FUNCTION_BLOCK MGE (* Composite Function Block Type *)
  (* Standard: 61499-2 *)
  (* Version 0.9, 12/05/2026, Medidor Geral de Energia. CAT top-level com 2 SYMLINKMULTIVARDST do tipo base Runtime.System.SYMLINKMULTIVARDST (sem hash - EAE expande pelo InterfaceParams). SYMLINKMULTIVARDST1 = 16xREAL (tensoes/correntes/pot ativa parcial+total/pot reativa parcial); SYMLINKMULTIVARDST2 = 4xREAL (pot reativa total/freq/FP/pot aparente total). *)
  PACKAGE Hidryco.HidrycoLib;
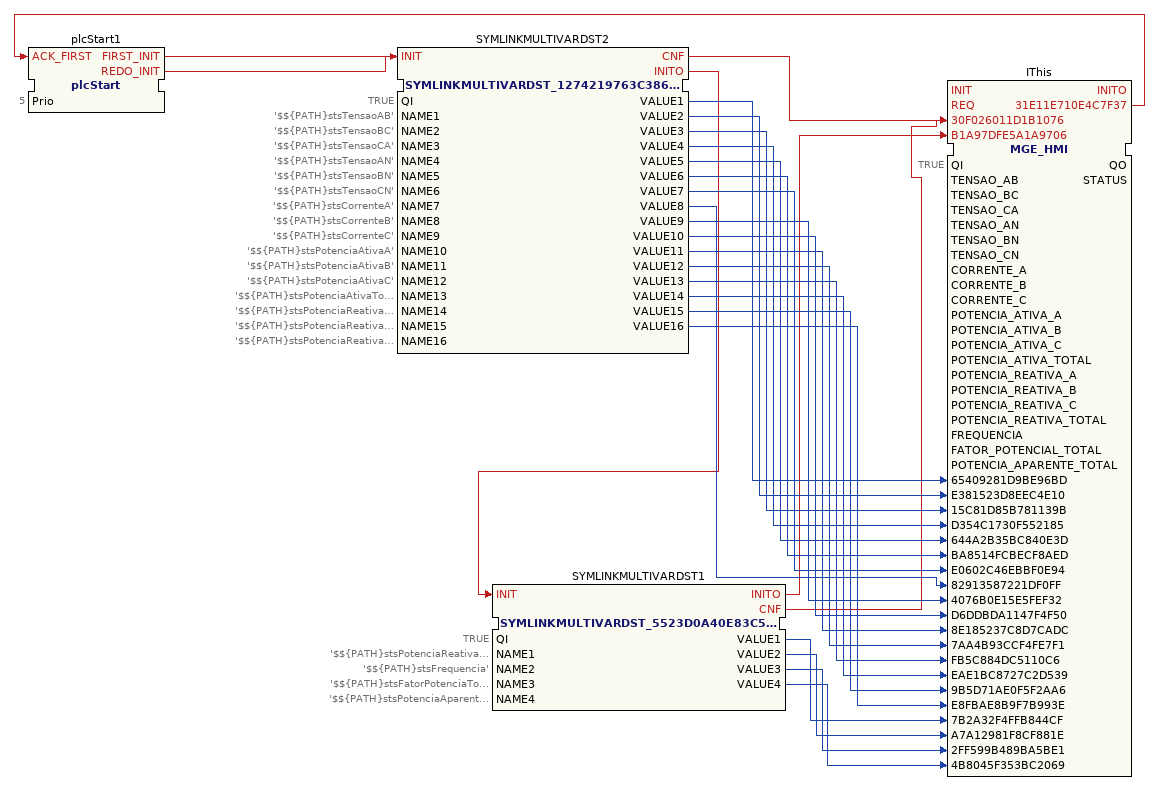
  FBS
    IThis : MGE_HMI(QI := TRUE);
    plcStart1 : plcStart(Prio := 5);
    SYMLINKMULTIVARDST2 : SYMLINKMULTIVARDST_1274219763C386EE8(QI := TRUE, NAME1 := '$${PATH}stsTensaoAB', NAME2 := '$${PATH}stsTensaoBC', NAME3 := '$${PATH}stsTensaoCA', NAME4 := '$${PATH}stsTensaoAN', NAME5 := '$${PATH}stsTensaoBN', NAME6 := '$${PATH}stsTensaoCN', NAME7 := '$${PATH}stsCorrenteA', NAME8 := '$${PATH}stsCorrenteB', NAME9 := '$${PATH}stsCorrenteC', NAME10 := '$${PATH}stsPotenciaAtivaA', NAME11 := '$${PATH}stsPotenciaAtivaB', NAME12 := '$${PATH}stsPotenciaAtivaC', NAME13 := '$${PATH}stsPotenciaAtivaTotal', NAME14 := '$${PATH}stsPotenciaReativaA', NAME15 := '$${PATH}stsPotenciaReativaB', NAME16 := '$${PATH}stsPotenciaReativaC'); {SET_ATTRIBUTE(Configuration.GenericFBType.InterfaceParams, Runtime.System#I:=16;VALUE${I$}:REAL,REAL,REAL,REAL,REAL,REAL,REAL,REAL,REAL,REAL,REAL,REAL,REAL,REAL,REAL,REAL)}
    SYMLINKMULTIVARDST1 : SYMLINKMULTIVARDST_5523D0A40E83C5C4(QI := TRUE, NAME1 := '$${PATH}stsPotenciaReativaTotal', NAME2 := '$${PATH}stsFrequencia', NAME3 := '$${PATH}stsFatorPotenciaTotal', NAME4 := '$${PATH}stsPotenciaAparenteTotal'); {SET_ATTRIBUTE(Configuration.GenericFBType.InterfaceParams, Runtime.System#I:=4;VALUE${I$}:REAL,REAL,REAL,REAL)}
  END_FBS
  EVENT_CONNECTIONS
    plcStart1.FIRST_INIT TO SYMLINKMULTIVARDST2.INIT;
    SYMLINKMULTIVARDST2.CNF TO IThis.30F026011D1B1076;
    IThis.31E11E710E4C7F37 TO plcStart1.ACK_FIRST;
    SYMLINKMULTIVARDST2.INITO TO SYMLINKMULTIVARDST1.INIT;
    SYMLINKMULTIVARDST1.INITO TO IThis.B1A97DFE5A1A9706;
    SYMLINKMULTIVARDST1.CNF TO IThis.30F026011D1B1076;
    plcStart1.REDO_INIT TO SYMLINKMULTIVARDST2.INIT;
  END_CONNECTIONS
  DATA_CONNECTIONS
    SYMLINKMULTIVARDST2.VALUE1 TO IThis.65409281D9BE96BD;
    SYMLINKMULTIVARDST2.VALUE2 TO IThis.E381523D8EEC4E10;
    SYMLINKMULTIVARDST2.VALUE3 TO IThis.15C81D85B781139B;
    SYMLINKMULTIVARDST2.VALUE4 TO IThis.D354C1730F552185;
    SYMLINKMULTIVARDST2.VALUE5 TO IThis.644A2B35BC840E3D;
    SYMLINKMULTIVARDST2.VALUE6 TO IThis.BA8514FCBECF8AED;
    SYMLINKMULTIVARDST2.VALUE7 TO IThis.E0602C46EBBF0E94;
    SYMLINKMULTIVARDST2.VALUE8 TO IThis.82913587221DF0FF;
    SYMLINKMULTIVARDST2.VALUE9 TO IThis.4076B0E15E5FEF32;
    SYMLINKMULTIVARDST2.VALUE10 TO IThis.D6DDBDA1147F4F50;
    SYMLINKMULTIVARDST2.VALUE11 TO IThis.8E185237C8D7CADC;
    SYMLINKMULTIVARDST2.VALUE12 TO IThis.7AA4B93CCF4FE7F1;
    SYMLINKMULTIVARDST2.VALUE13 TO IThis.FB5C884DC5110C6;
    SYMLINKMULTIVARDST2.VALUE14 TO IThis.EAE1BC8727C2D539;
    SYMLINKMULTIVARDST2.VALUE15 TO IThis.9B5D71AE0F5F2AA6;
    SYMLINKMULTIVARDST2.VALUE16 TO IThis.E8FBAE8B9F7B993E;
    SYMLINKMULTIVARDST1.VALUE1 TO IThis.7B2A32F4FFB844CF;
    SYMLINKMULTIVARDST1.VALUE2 TO IThis.A7A12981F8CF881E;
    SYMLINKMULTIVARDST1.VALUE3 TO IThis.2FF599B489BA5BE1;
    SYMLINKMULTIVARDST1.VALUE4 TO IThis.4B8045F353BC2069;
  END_CONNECTIONS
END_FUNCTION_BLOCK
